# EPICS IOC start-up script: iocsh/digitelPump_D500.iocsh
asynSetOption("$(PORT)", -1, "baud",    "9600")
asynSetOption("$(PORT)", -1, "bits",    "7")
asynSetOption("$(PORT)", -1, "stop",    "1")
asynSetOption("$(PORT)", -1, "parity",  "even")
asynSetOption("$(PORT)", -1, "clocal",  "Y")
asynSetOption("$(PORT)", -1, "crtscts", "N")
asynOctetSetInputEos( "$(PORT)", -1, "\n\r")
asynOctetSetOutputEos("$(PORT)", -1, "\r")

dbLoadRecords("$(VAC)/vacApp/Db/digitelPump.db", "P=$(PREFIX),PUMP=$(INSTANCE),PORT=$(PORT),ADDR=$(ADDR=0),DEV=D500,STN=$(STN=1)")
